PROGRAM P_Demo_PBOOL_TO_BOOL
VAR
    xRealValue           : BOOL := TRUE; // 模拟 wire 缓冲区中的 BOOL 字段
    pBOOLField           : POINTER TO BOOL; // 业务侧先算好的字段地址（ADR 或 pBase+nOff）
    bExtractField        : BOOL; // 在线置 TRUE 触发一次解析
    xRealValue_extracted : BOOL; // 解析后的副本，供业务逻辑使用
END_VAR

// ============================================================
// Tc2_Utilities.PBOOL_TO_BOOL 演示程序（FUNCTION）
// ============================================================
// 场景：从一段二进制 wire 缓冲区里按偏移取 BOOL 字段（Modbus/CAN/ADS Raw）。
// 价值：替代手写 pField + nOff + ^ 指针算术；一次调用取值，少打错符号。
// 验证：在线写 xRealValue := TRUE；bExtractField := TRUE；
//       下一周期 xRealValue_extracted 应等于 xRealValue。
// ============================================================

// 业务代码通常已经算好字段地址（pBase + 协议偏移）；演示用 ADR 等价
pBOOLField := ADR(xRealValue);

IF bExtractField AND pBOOLField <> 0 THEN
    // 单次完整调用：避免手写 ^ 解引用，统一风格便于和字节序转换串联
    xRealValue_extracted := PBOOL_TO_BOOL(pBOOLField);
    bExtractField := FALSE;
END_IF;

END_PROGRAM

(* stored: Version 1.1.0.1, ProductVersion 3.1.4024.5
   POU P_Demo_PBOOL_TO_BOOL: Id {9cd7e64c-a88d-5d0f-a0b4-37386362107b}, SpecialFunc None *)
